PROGRAM CallHardware

//conveyors
pushConveyorsToArray();
callConveyors();

//robots
robot1();
robot2();
robot3();
robot4();
//robot5();
//robot6();

//A23
wrapperA23();

//A22
skidA22Left();
skidA22Right();
magazineA22Left();
magazineA22Right();

insertionA22Left(
	enable:= TRUE, 
	slider:= verticalDriveA22Left, 
	screw:= horizontalDriveA22Left, 
	contact=> , 
	active=> , 
	error=> , 
	home=> , 
	homingComplete=> , 
	sliderPos=> );
	
insertionA22Right(
	enable:= TRUE, 
	slider:= verticalDriveA22Right, 
	screw:= horizontalDriveA22Right, 
	contact=> , 
	active=> , 
	error=> , 
	home=> , 
	homingComplete=> , 
	sliderPos=> );
	
pistonA22Bottom();
wrapperA22();

//A21
skidA21Left();
skidA21Right();

magazineA21Left();
magazineA21Right();

stagingTableLeft();
stagingTableRight();

strapperA21();

insertionA21Left(
	enable:= TRUE, 
	slider:= verticalDriveA21Left, 
	screw:= horizontalDriveA21Left, 
	contact=> , 
	active=> , 
	error=> , 
	home=> , 
	homingComplete=> , 
	sliderPos=> );
	
insertionA21Right(
	enable:= TRUE, 
	slider:= verticalDriveA21Right, 
	screw:= horizontalDriveA21Right, 
	contact=> , 
	active=> , 
	error=> , 
	home=> , 
	homingComplete=> , 
	sliderPos=> );
	
pistonA21Bottom();

METHOD PRIVATE callConveyors : BOOL
VAR
	i : DINT;
END_VAR
//rewrite this method, call every conveyor individually
//calling via loop will not call derived implementations
(*
FOR i:=1 TO numConveyors BY 1 DO
	conveyorsArr[i]^(
		bEnable:= , 
		enable=> , 
		direction=> , 
		pulse=> , 
		reset=> , 
		error=> , 
		sensorEntry=> , 
		sensorExit=> , 
		requestLifter=> , 
		lifterEnable=> , 
		lifterDirection=> , 
		lifterPulse=> , 
		lifterReset=> , 
		lifterError=> , 
		extended=> , 
		retracted=> , 
		position=> , 
		velocity=> );
END_FOR
*)
END_METHOD

METHOD PRIVATE pushConveyorsToArray : BOOL
conveyorsArr[1] := ADR(A24_SC_C01);
conveyorsArr[2] := ADR(A24_LRC_C02);
conveyorsArr[3] := ADR(A24_SC_C03);
conveyorsArr[4] := ADR(A24_LRC_C04);
conveyorsArr[5] := ADR(A24_SC_C05);
conveyorsArr[6] := ADR(A24_LRC_C06);
conveyorsArr[7] := ADR(A24_SC_C07);
conveyorsArr[8] := ADR(A24_LRC_C08);
conveyorsArr[9] := ADR(A24_SC_C09);
conveyorsArr[10] := ADR(A24_LRC_C10);
conveyorsArr[11] := ADR(A24_SC_C11);
conveyorsArr[12] := ADR(A24_LRC_C12);
conveyorsArr[13] := ADR(A24_SC_C13);

conveyorsArr[14] := ADR(A23_LSC_C14);

conveyorsArr[15] := ADR(A22_SC_C15);
conveyorsArr[16] := ADR(A22_LSC_C16);
conveyorsArr[17] := ADR(A22_LSC_C17);

conveyorsArr[18] := ADR(A21_SC_C18);
conveyorsArr[19] := ADR(A21_LSC_C19);
conveyorsArr[20] := ADR(A21_LSC_C20);
conveyorsArr[21] := ADR(A21_LSC_C21);

conveyorsArr[22] := ADR(A25_SC_C22);
conveyorsArr[23] := ADR(A25_LSC_C23);
conveyorsArr[24] := ADR(A25_SC_C24);
conveyorsArr[25] := ADR(A25_LSLCC_C25);
conveyorsArr[26] := ADR(A25_SC_C26);
conveyorsArr[27] := ADR(A25_LSLCC_C27);
conveyorsArr[28] := ADR(A25_SC_C28);
conveyorsArr[29] := ADR(A25_LSC_C29);
conveyorsArr[30] := ADR(A25_SC_C30);
conveyorsArr[31] := ADR(A25_SC_C31);
conveyorsArr[32] := ADR(A25_SC_C32);
conveyorsArr[33] := ADR(A25_SC_C33);
conveyorsArr[34] := ADR(A25_SC_C34);
conveyorsArr[35] := ADR(A25_SC_C35);
conveyorsArr[36] := ADR(A25_SC_C36);
conveyorsArr[37] := ADR(A25_SC_C37);
conveyorsArr[38] := ADR(A25_SC_C38);
END_METHOD

END_PROGRAM

(* stored: Version 1.1.0.1, ProductVersion 3.1.4024.11
   POU CallHardware: Id {37cad5aa-fa76-4d83-b429-cad99db8cb21}, SpecialFunc None
   Method callConveyors: Id {365141b1-cb20-44d4-87c7-77ba15ac296c}
   Method pushConveyorsToArray: Id {cb74d2be-b24d-425a-bc95-cdcd1fdaeaaf} *)
